// TIA Portal V20 export
// export: Created 2025-12-01T14:57:32.5687977Z, ExportSetting None, DisplayName Totally Integrated Automation Portal, DisplayVersion V20 Update 3, DisplayName TIA Portal Openness, DisplayVersion V20 Update 3, DisplayName TIA Portal Version Control Interface, DisplayVersion V20 Update 3, DisplayName STEP 7 Professional, DisplayVersion V20 Update 3, DisplayName STEP 7 Safety, DisplayVersion V20 Update 2, DisplayName WinCC Basic/Comfort/Advanced, DisplayVersion V20 Update 3, DisplayName WinCC Professional, DisplayVersion V20 Update 3, DisplayName WinCC Unified, DisplayVersion V20 Update 3
DATA_BLOCK "DB951_InterlockMaquinas"   // DB951
{ S7_Optimized_Access := 'FALSE' }
// stored: AutoNumber false
   VAR
      Maquina : Array[0..15] of Struct
         PosOK : Bool;
         Mesa_Origen : UInt;
         Mesa_Destino : UInt;
         Derecha : Bool;
         Izquierda : Bool;
         H1 : Struct
            In : "UDT_MesaMaquina_Interlock";
            Out { S7_SetPoint := 'True'} : "UDT_MesaMaquina_Interlock";
            Mesa_EntradaDerecha { S7_SetPoint := 'True'} : UInt;
            Mesa_EntradaIzquierda : UInt;
         END_STRUCT;
         H2 : Struct
            In : "UDT_MesaMaquina_Interlock";
            Out { S7_SetPoint := 'True'} : "UDT_MesaMaquina_Interlock";
            Mesa_EntradaDerecha { S7_SetPoint := 'True'} : UInt;
            Mesa_EntradaIzquierda { S7_SetPoint := 'True'} : UInt;
         END_STRUCT;
         Mesa : Array[0..500] of Struct
            In : "UDT_MesaAcometida_Interlock";
            Out : "UDT_MesaAcometida_Interlock";
            PeticionPos : Bool;
            PosOK_H1 : Bool;
            PosOK_H2 : Bool;
            MesaEntrada { S7_SetPoint := 'True'} : UInt;
         END_STRUCT;
      END_STRUCT;
   END_VAR
BEGIN
   Maquina[1].Mesa[1..11].PeticionPos := false;
   Maquina[3].Mesa[2..8].PeticionPos := false;
   Maquina[3].Mesa[10..11].PeticionPos := false;
   Maquina[1].Mesa[1..11].PosOK_H1 := false;
   Maquina[3].Mesa[2..8].PosOK_H1 := false;
   Maquina[3].Mesa[10..11].PosOK_H1 := false;
END_DATA_BLOCK
